// Mitsubishi GX Works2 project: 通信テスト用   PLC: FX3U/FX3UC

PROGRAM MAIN
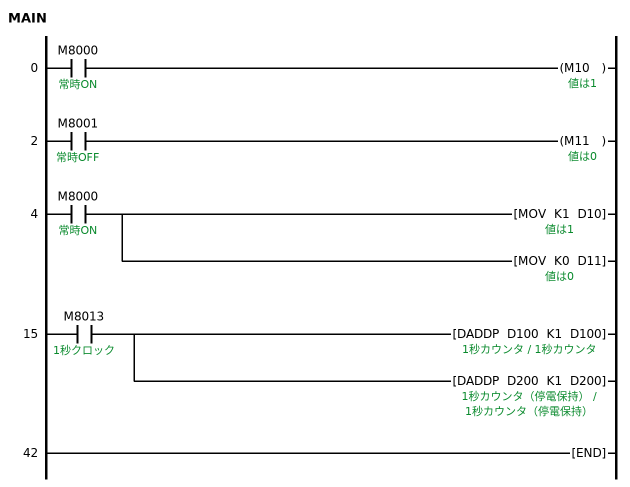
0     LD      M8000  ; 常時ON
      OUT     M10  ; 値は1
2     LD      M8001  ; 常時OFF
      OUT     M11  ; 値は0
4     LD      M8000  ; 常時ON
      MOV     K1 D10  ; 値は1
      MOV     K0 D11  ; 値は0
15    LD      M8013  ; 1秒クロック
      DADDP   D100 K1 D100  ; 1秒カウンタ
      DADDP   D200 K1 D200  ; 1秒カウンタ（停電保持）
42    END
END_PROGRAM
